FUNCTION_BLOCK Q_Attribute (* Command change attribute( Part 6 - F.38 ) *)
  (* Standard: ISO 11783-6; Description: Copyright (c) 2022 HR Agrartechnik GmbH This program and the accompanying materials are made available under the terms of the Eclipse Public License 2.0 which is available at https://www.eclipse.org/legal/epl-2.0/ SPDX-License-Identifier: EPL-2.0 see Description Tab *)
  (* Version 1.0, 2022-07-08, Franz Höpfinger, HR Agrartechnik GmbH *)
  PACKAGE isobus::UT::Q;
  IMPORT isobus::UT::Q::const::IDs::ID_NULL;
  (* Documentation:
  Command change attribute ( Part 6 - F.38 )
   This command is used to change any attribute with an assigned AID. This message cannot be used to change strings. It addresses two distinct parameters with different validity rules each — u16ObjId (the object whose attribute is changed) and u8IdAttribute (the Attribute ID, AID, selecting the attribute).
   Valid values for u16ObjId (the object whose attribute is changed)
   An attribute Object ID is valid if it falls within one of the following ISO 11783-6 ID ranges (Annex F.38):
    - DataMask: 1000 – 1999
   - AlarmMask: 2000 – 2999
   - SoftKeyMask: 4000 – 4999
   - Key: 5000 – 5999
   - Button: 6000 – 6999
   - InputBooleanField: 7000 – 7999
   - InputStringField: 8000 – 8999
   - InputNumberField: 9000 – 9999
   - InputListField: 10000 – 10999
   - AuxiliaryFunctionType2: 31000 – 31999
    Valid values for u8IdAttribute (AID)
   The Attribute ID (AID) selects which attribute of the addressed object is changed. Valid AIDs are object-type specific and are defined in ISO 11783-6 Annex B, in the attribute table of each object type. An AID with no attribute assigned is rejected by the VT (F.39, bit 1 = Invalid Attribute ID). The new value is transmitted little endian in bytes 5–8 of the command (F.38) — this FB passes it as u32ValueAttribute.
   ID_NULL (65535) is not a command target but can be used in INIT to deactivate the FB. Any ID outside these ranges is invalid for commanding.
   Activate / Deactivate
   The FB is deactivated by default. It becomes active when INIT provides a valid attribute Object ID. Sending INIT with ID_NULL (65535) deactivates the FB again. This toggle can be repeated arbitrarily.
    - INIT + ID_NULL (65535): FB deactivated, STATUS="DEACTIVATED", s16result=VT_E_DEACTIVATED (-40)
   - INIT + valid attribute ID: FB activated, STATUS="initialized", s16result=VT_E_NO_ERR (0). If a REQ was buffered before, it is executed immediately.
   - INIT + invalid ID: STATUS="ERROR: Invalid Object ID (not an attribute object)", s16result=VT_E_INVALID_OBJECT_ID (-132)
    REQ Handling
    - REQ before any INIT: Buffered, STATUS="Buffered: INIT not yet completed", s16result=VT_E_NOT_READY (-131)
   - REQ while deactivated (INIT came with NULL or invalid ID): STATUS shows the actual deactivation reason, s16result=VT_E_DEACTIVATED (-40) or VT_E_INVALID_OBJECT_ID (-132)
   - REQ while active: Command sent to VT, result reflected in CNF
    param[in] {u16ObjId, uint16_t}
   Object ID. Use ID_NULL (65535) to deactivate the FB. Use a valid attribute object ID to activate.
   param[in] {u8IdAttribute, uint8_t}
   Attribute ID (AID) - see description of wished object
   param[in] {u32ValueAttribute, uint32_t}
   New value for attribute
   Return Values (s16result):
   int16_t
    - VT_E_NO_ERR (0) - OK
   - VT_E_DEACTIVATED (-40) - FB deactivated (INIT received with ID_NULL)
   - VT_E_INVALID_OBJECT_ID (-132) - Object ID is invalid (not an attribute object)
   - VT_E_NOT_READY (-131) - Buffered: INIT not yet completed
   - VT_E_OVERFLOW (-6) - buffer overflow
   - VT_E_NOACT (-8) - Command not possible in current state
   - VT_E_NO_INSTANCE (-21) - No VT client available
   - VT_E_ISO_INSTANCE_INVALID (-129) - Identifier for instance (connection) invalid
   - VT_E_NOT_ALIVE (-130) - Identifier for instance valid, but VT Dead.
    Instanz-Eindeutigkeit (Instance Uniqueness)
   Dieser Baustein erfordert Instanz-Eindeutigkeit bezüglich des Paares (u16ObjId, u8IdAttribute). Es darf im gesamten Programm nur eine Instanz von Q_Attribute für dasselbe Objekt-Attribut-Paar existieren. Eine zweite Instanz auf dieselbe Objekt-ID und Attribut-ID wird bei INIT deaktiviert (STATUS = "This objID is already in use").
  *)
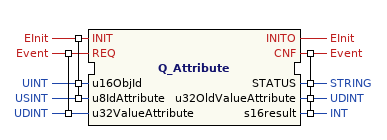
  EVENT_INPUT
    INIT : EInit WITH u16ObjId, u8IdAttribute; (* Service Initialization *)
    REQ WITH u32ValueAttribute; (* Service Request *)
  END_EVENT
  EVENT_OUTPUT
    INITO : EInit; (* Initialization Confirm *)
    CNF WITH STATUS, u32OldValueAttribute, s16result; (* Confirmation of Requested Service *)
  END_EVENT
  VAR_INPUT
    u16ObjId : UINT := ID_NULL; (* Object ID *)
    u8IdAttribute : USINT; (* Attribute ID (AID) - see description of wished object *)
    u32ValueAttribute : UDINT; (* New value for attribute *)
  END_VAR
  VAR_OUTPUT
    STATUS : STRING; (* Service Status *)
    u32OldValueAttribute : UDINT; (* Old value for attribute *)
    s16result : INT; (* retval see description *)
  END_VAR
END_FUNCTION_BLOCK
